// TwinCAT 3 PLC project main
// ProgramVersion: 3.1.4024.0
// libraries:
//   Tc2_Standard, * (Beckhoff Automation GmbH)
//   Tc2_System, * (Beckhoff Automation GmbH)
//   Tc3_Module, * (Beckhoff Automation GmbH)
// project tree:
//   / GlobalTextList.TcGTLO, PlcTask.TcTTO, Visualization Manager.TcVMO (not stored)
//   POUs/ MAIN.TcPOU
//   VISUs/ Visu.TcVIS

CONFIGURATION main
    RESOURCE PLC ON TwinCAT3
        TASK PlcTask(INTERVAL := T#10ms, PRIORITY := 20);
        PROGRAM MAIN WITH PlcTask : MAIN;
    END_RESOURCE
END_CONFIGURATION

// ---- POUs/MAIN.TcPOU
PROGRAM MAIN
VAR
	bInput : BOOL;
	bOutput : BOOL;
END_VAR

bOutput := bInput;

END_PROGRAM

// ---- VISUs/Visu.TcVIS
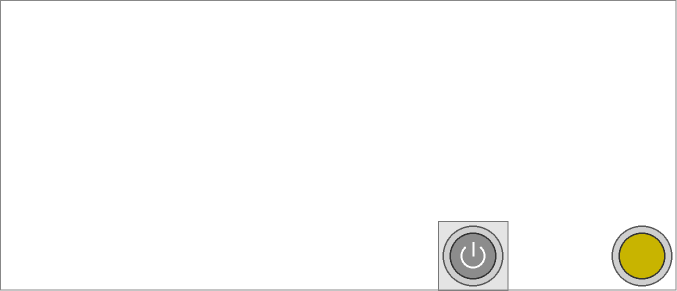
VISUALIZATION Visu  // 677x291
    PowerSwitch (438,221 70x70), variable: MAIN.bInput, behaviour: TOGGLE, style: Switch-PowerSwitch-Gray
    Lamp1 (607,221 70x70), variable: MAIN.bOutput, style: Lamp-Lamp1-Yellow
END_VISUALIZATION
